// Mitsubishi GX Developer project: 12-1008_20141007   PLC: FX3U

PROGRAM MAIN
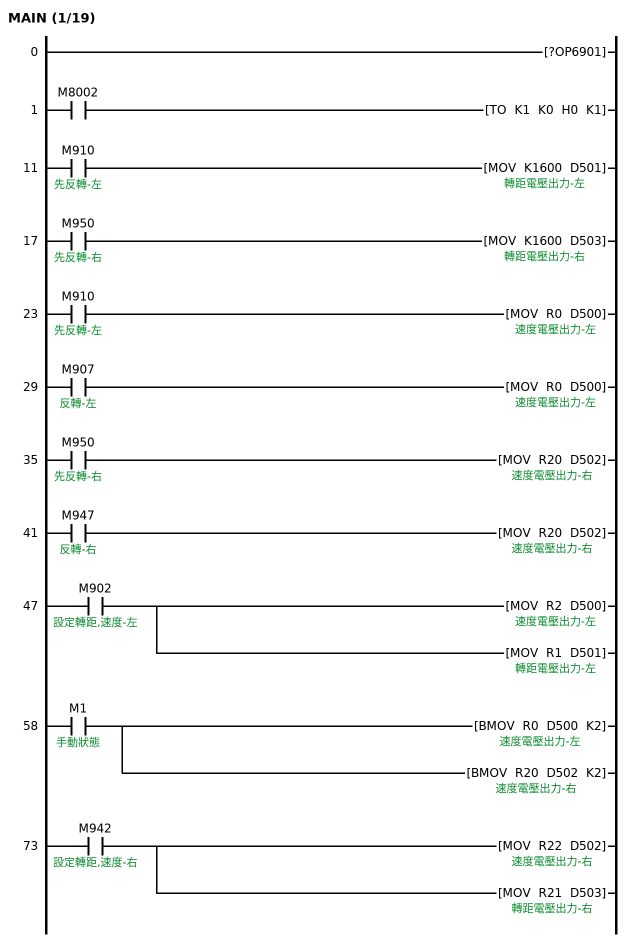
0     ?OP6901
1     LD      M8002
      TO      K1 K0 H0 K1
11    LD      M910  ; 先反轉-左
      MOV     K1600 D501  ; 轉距電壓出力-左
17    LD      M950  ; 先反轉-右
      MOV     K1600 D503  ; 轉距電壓出力-右
23    LD      M910  ; 先反轉-左
      MOV     R0 D500  ; 速度電壓出力-左
29    LD      M907  ; 反轉-左
      MOV     R0 D500
35    LD      M950  ; 先反轉-右
      MOV     R20 D502  ; 速度電壓出力-右
41    LD      M947  ; 反轉-右
      MOV     R20 D502
47    LD      M902  ; 設定轉距,速度-左
      MOV     R2 D500
      MOV     R1 D501
58    LD      M1  ; 手動狀態
      BMOV    R0 D500 K2
      BMOV    R20 D502 K2
73    LD      M942  ; 設定轉距,速度-右
      MOV     R22 D502
      MOV     R21 D503
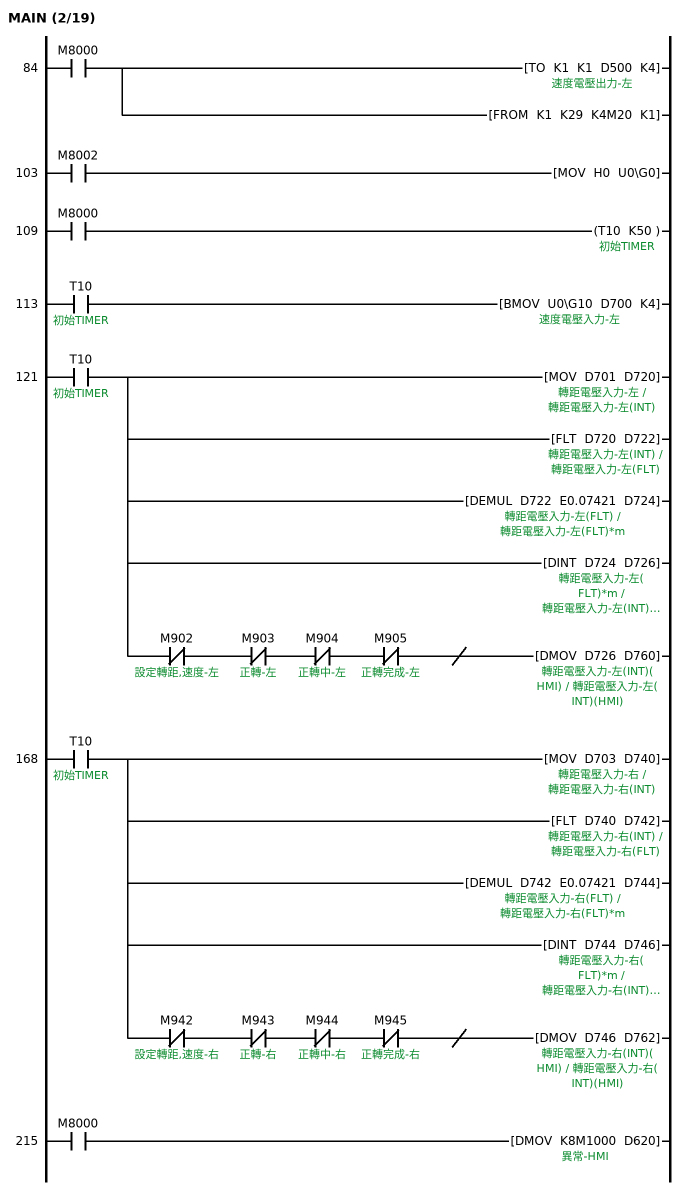
84    LD      M8000
      TO      K1 K1 D500 K4
      FROM    K1 K29 K4M20 K1  ; DA模組狀態
103   LD      M8002
      MOV     H0 U0\G0
109   LD      M8000
      OUT     T10 K50  ; 初始TIMER
113   LD      T10  ; 初始TIMER
      BMOV    U0\G10 D700 K4  ; 速度電壓入力-左
121   LD      T10  ; 初始TIMER
      MOV     D701 D720  ; 轉距電壓入力-左 / 轉距電壓入力-左(INT)
      FLT     D720 D722  ; 轉距電壓入力-左(FLT)
      DEMUL   D722 E0.07421 D724  ; 轉距電壓入力-左(FLT)*m
      DINT    D724 D726  ; 轉距電壓入力-左(INT)(HMI)
      ANI     M902  ; 設定轉距,速度-左
      ANI     M903  ; 正轉-左
      ANI     M904  ; 正轉中-左
      ANI     M905  ; 正轉完成-左
      INV
      DMOV    D726 D760  ; 轉距電壓入力-左(INT)(HMI)
168   LD      T10  ; 初始TIMER
      MOV     D703 D740  ; 轉距電壓入力-右 / 轉距電壓入力-右(INT)
      FLT     D740 D742  ; 轉距電壓入力-右(FLT)
      DEMUL   D742 E0.07421 D744  ; 轉距電壓入力-右(FLT)*m
      DINT    D744 D746  ; 轉距電壓入力-右(INT)(HMI)
      ANI     M942  ; 設定轉距,速度-右
      ANI     M943  ; 正轉-右
      ANI     M944  ; 正轉中-右
      ANI     M945  ; 正轉完成-右
      INV
      DMOV    D746 D762  ; 轉距電壓入力-右(INT)(HMI)
215   LD      M8000
      DMOV    K8M1000 D620  ; 滿料異常 / 異常-HMI
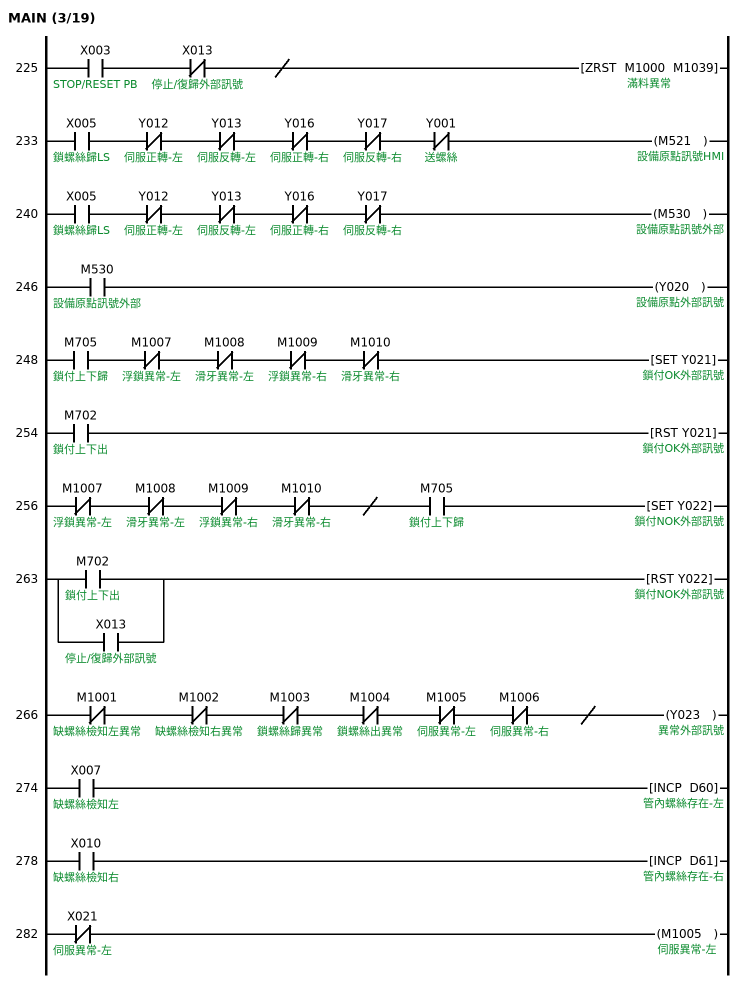
225   LD      X003  ; STOP/RESET PB
      ANI     X013  ; 停止/復歸外部訊號
      INV
      ZRST    M1000 M1039
233   LD      X005  ; 鎖螺絲歸LS
      ANI     Y012  ; 伺服正轉-左
      ANI     Y013  ; 伺服反轉-左
      ANI     Y016  ; 伺服正轉-右
      ANI     Y017  ; 伺服反轉-右
      ANI     Y001  ; 送螺絲
      OUT     M521  ; 設備原點訊號HMI
240   LD      X005  ; 鎖螺絲歸LS
      ANI     Y012  ; 伺服正轉-左
      ANI     Y013  ; 伺服反轉-左
      ANI     Y016  ; 伺服正轉-右
      ANI     Y017  ; 伺服反轉-右
      OUT     M530  ; 設備原點訊號外部
246   LD      M530  ; 設備原點訊號外部
      OUT     Y020  ; 設備原點外部訊號
248   LD      M705  ; 鎖付上下歸
      ANI     M1007  ; 浮鎖異常-左
      ANI     M1008  ; 滑牙異常-左
      ANI     M1009  ; 浮鎖異常-右
      ANI     M1010  ; 滑牙異常-右
      SET     Y021  ; 鎖付OK外部訊號
254   LD      M702  ; 鎖付上下出
      RST     Y021  ; 鎖付OK外部訊號
256   LDI     M1007  ; 浮鎖異常-左
      ANI     M1008  ; 滑牙異常-左
      ANI     M1009  ; 浮鎖異常-右
      ANI     M1010  ; 滑牙異常-右
      INV
      AND     M705  ; 鎖付上下歸
      SET     Y022  ; 鎖付NOK外部訊號
263   LD      M702  ; 鎖付上下出
      OR      X013  ; 停止/復歸外部訊號
      RST     Y022  ; 鎖付NOK外部訊號
266   LDI     M1001  ; 缺螺絲檢知左異常
      ANI     M1002  ; 缺螺絲檢知右異常
      ANI     M1003  ; 鎖螺絲歸異常
      ANI     M1004  ; 鎖螺絲出異常
      ANI     M1005  ; 伺服異常-左
      ANI     M1006  ; 伺服異常-右
      INV
      OUT     Y023  ; 異常外部訊號
274   LD      X007  ; 缺螺絲檢知左
      INCP    D60  ; 管內螺絲存在-左
278   LD      X010  ; 缺螺絲檢知右
      INCP    D61  ; 管內螺絲存在-右
282   LDI     X021  ; 伺服異常-左
      OUT     M1005  ; 伺服異常-左
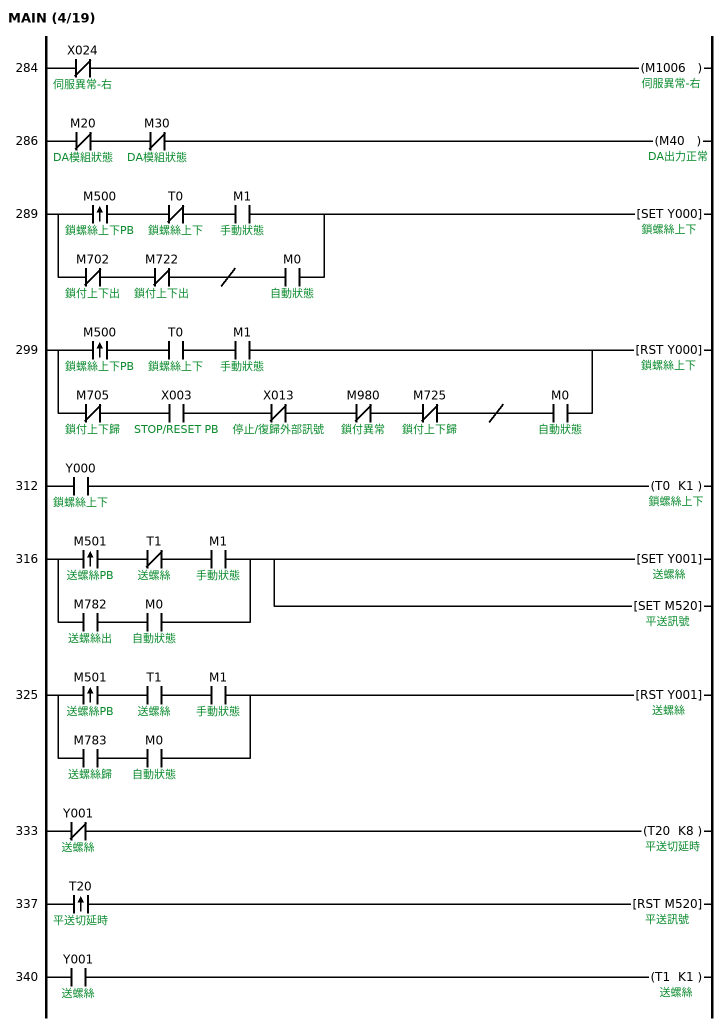
284   LDI     X024  ; 伺服異常-右
      OUT     M1006  ; 伺服異常-右
286   LDI     M20  ; DA模組狀態
      ANI     M30  ; DA模組狀態
      OUT     M40  ; DA出力正常
289   LDP     M500  ; 鎖螺絲上下PB
      ANI     T0  ; 鎖螺絲上下
      AND     M1  ; 手動狀態
      LDI     M702  ; 鎖付上下出
      ANI     M722  ; 鎖付上下出
      INV
      AND     M0  ; 自動狀態
      ORB
      SET     Y000  ; 鎖螺絲上下
299   LDP     M500  ; 鎖螺絲上下PB
      AND     T0  ; 鎖螺絲上下
      AND     M1  ; 手動狀態
      LDI     M705  ; 鎖付上下歸
      AND     X003  ; STOP/RESET PB
      ANI     X013  ; 停止/復歸外部訊號
      ANI     M980  ; 鎖付異常
      ANI     M725  ; 鎖付上下歸
      INV
      AND     M0  ; 自動狀態
      ORB
      RST     Y000  ; 鎖螺絲上下
312   LD      Y000  ; 鎖螺絲上下
      OUT     T0 K1  ; 鎖螺絲上下
316   LDP     M501  ; 送螺絲PB
      ANI     T1  ; 送螺絲
      AND     M1  ; 手動狀態
      LD      M782  ; 送螺絲出
      AND     M0  ; 自動狀態
      ORB
      SET     Y001  ; 送螺絲
      SET     M520  ; 平送訊號
325   LDP     M501  ; 送螺絲PB
      AND     T1  ; 送螺絲
      AND     M1  ; 手動狀態
      LD      M783  ; 送螺絲歸
      AND     M0  ; 自動狀態
      ORB
      RST     Y001  ; 送螺絲
333   LDI     Y001  ; 送螺絲
      OUT     T20 K8  ; 平送切延時
337   LDP     T20  ; 平送切延時
      RST     M520  ; 平送訊號
340   LD      Y001  ; 送螺絲
      OUT     T1 K1  ; 送螺絲
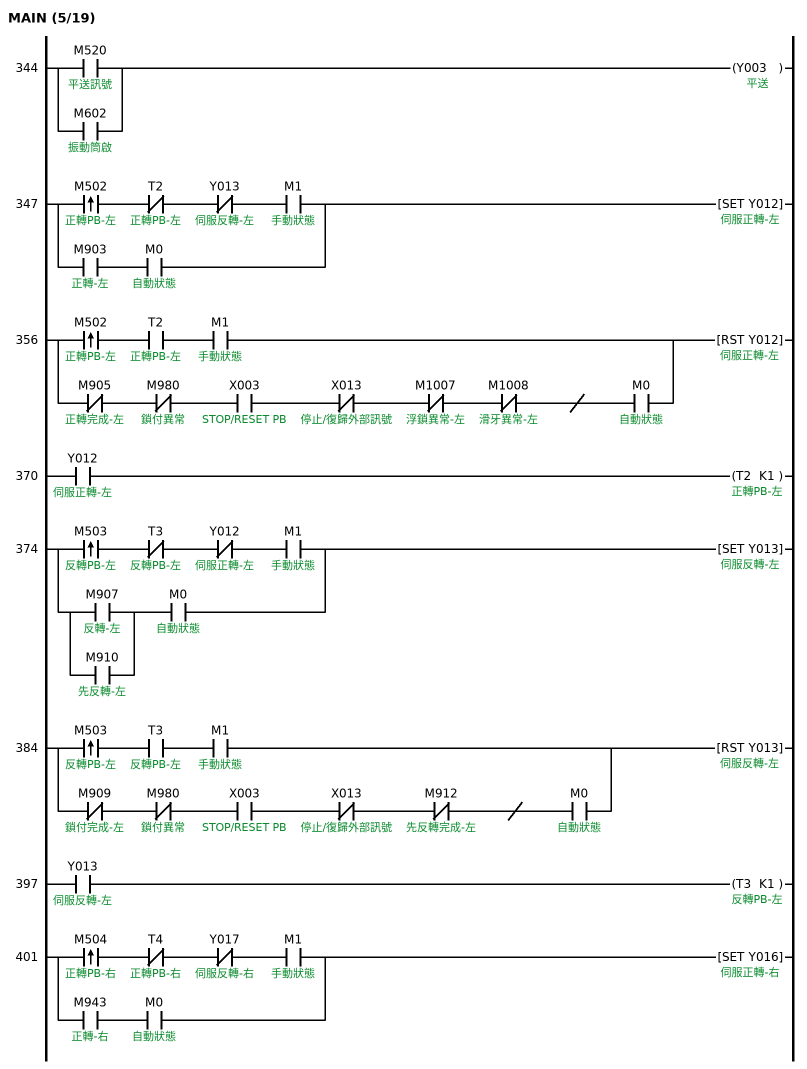
344   LD      M520  ; 平送訊號
      OR      M602  ; 振動筒啟
      OUT     Y003  ; 平送
347   LDP     M502  ; 正轉PB-左
      ANI     T2  ; 正轉PB-左
      ANI     Y013  ; 伺服反轉-左
      AND     M1  ; 手動狀態
      LD      M903  ; 正轉-左
      AND     M0  ; 自動狀態
      ORB
      SET     Y012  ; 伺服正轉-左
356   LDP     M502  ; 正轉PB-左
      AND     T2  ; 正轉PB-左
      AND     M1  ; 手動狀態
      LDI     M905  ; 正轉完成-左
      ANI     M980  ; 鎖付異常
      AND     X003  ; STOP/RESET PB
      ANI     X013  ; 停止/復歸外部訊號
      ANI     M1007  ; 浮鎖異常-左
      ANI     M1008  ; 滑牙異常-左
      INV
      AND     M0  ; 自動狀態
      ORB
      RST     Y012  ; 伺服正轉-左
370   LD      Y012  ; 伺服正轉-左
      OUT     T2 K1  ; 正轉PB-左
374   LDP     M503  ; 反轉PB-左
      ANI     T3  ; 反轉PB-左
      ANI     Y012  ; 伺服正轉-左
      AND     M1  ; 手動狀態
      LD      M907  ; 反轉-左
      OR      M910  ; 先反轉-左
      AND     M0  ; 自動狀態
      ORB
      SET     Y013  ; 伺服反轉-左
384   LDP     M503  ; 反轉PB-左
      AND     T3  ; 反轉PB-左
      AND     M1  ; 手動狀態
      LDI     M909  ; 鎖付完成-左
      ANI     M980  ; 鎖付異常
      AND     X003  ; STOP/RESET PB
      ANI     X013  ; 停止/復歸外部訊號
      ANI     M912  ; 先反轉完成-左
      INV
      AND     M0  ; 自動狀態
      ORB
      RST     Y013  ; 伺服反轉-左
397   LD      Y013  ; 伺服反轉-左
      OUT     T3 K1  ; 反轉PB-左
401   LDP     M504  ; 正轉PB-右
      ANI     T4  ; 正轉PB-右
      ANI     Y017  ; 伺服反轉-右
      AND     M1  ; 手動狀態
      LD      M943  ; 正轉-右
      AND     M0  ; 自動狀態
      ORB
      SET     Y016  ; 伺服正轉-右
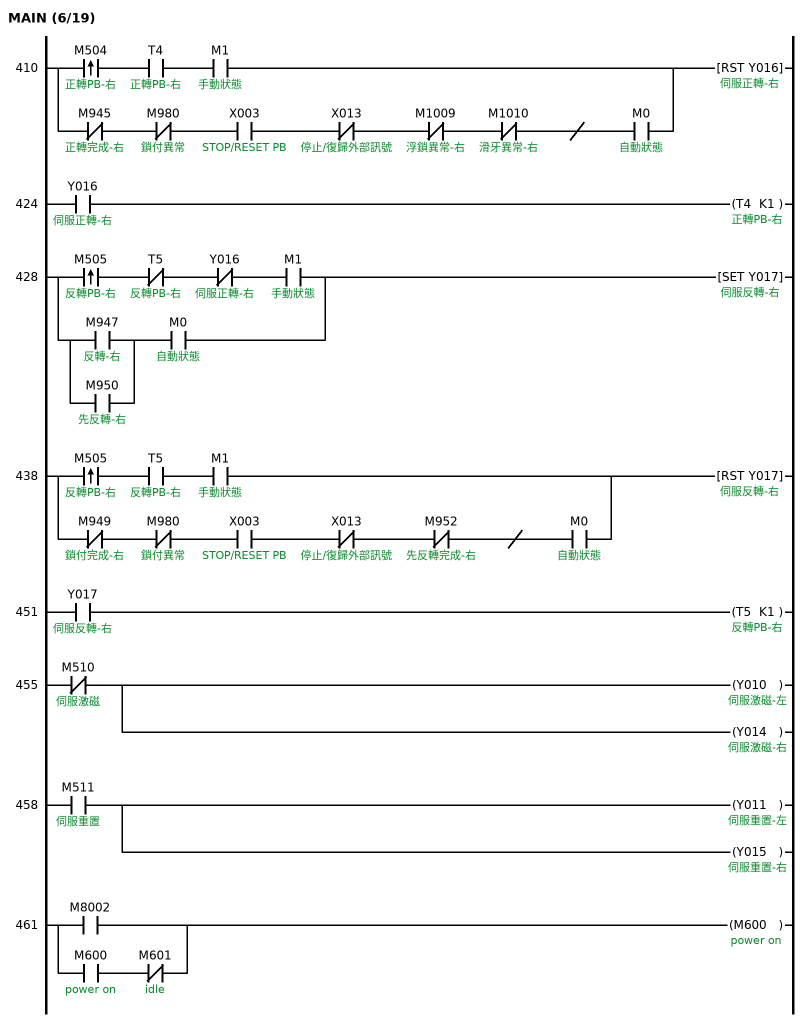
410   LDP     M504  ; 正轉PB-右
      AND     T4  ; 正轉PB-右
      AND     M1  ; 手動狀態
      LDI     M945  ; 正轉完成-右
      ANI     M980  ; 鎖付異常
      AND     X003  ; STOP/RESET PB
      ANI     X013  ; 停止/復歸外部訊號
      ANI     M1009  ; 浮鎖異常-右
      ANI     M1010  ; 滑牙異常-右
      INV
      AND     M0  ; 自動狀態
      ORB
      RST     Y016  ; 伺服正轉-右
424   LD      Y016  ; 伺服正轉-右
      OUT     T4 K1  ; 正轉PB-右
428   LDP     M505  ; 反轉PB-右
      ANI     T5  ; 反轉PB-右
      ANI     Y016  ; 伺服正轉-右
      AND     M1  ; 手動狀態
      LD      M947  ; 反轉-右
      OR      M950  ; 先反轉-右
      AND     M0  ; 自動狀態
      ORB
      SET     Y017  ; 伺服反轉-右
438   LDP     M505  ; 反轉PB-右
      AND     T5  ; 反轉PB-右
      AND     M1  ; 手動狀態
      LDI     M949  ; 鎖付完成-右
      ANI     M980  ; 鎖付異常
      AND     X003  ; STOP/RESET PB
      ANI     X013  ; 停止/復歸外部訊號
      ANI     M952  ; 先反轉完成-右
      INV
      AND     M0  ; 自動狀態
      ORB
      RST     Y017  ; 伺服反轉-右
451   LD      Y017  ; 伺服反轉-右
      OUT     T5 K1  ; 反轉PB-右
455   LDI     M510  ; 伺服激磁
      OUT     Y010  ; 伺服激磁-左
      OUT     Y014  ; 伺服激磁-右
458   LD      M511  ; 伺服重置
      OUT     Y011  ; 伺服重置-左
      OUT     Y015  ; 伺服重置-右
461   LD      M8002
      LD      M600  ; power on
      ANI     M601  ; idle
      ORB
      OUT     M600  ; power on
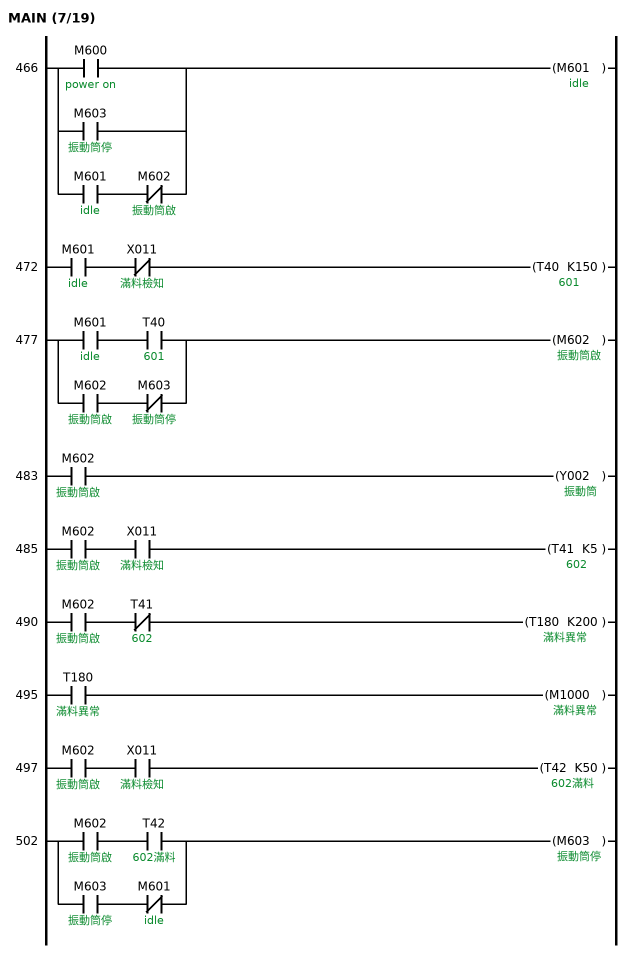
466   LD      M600  ; power on
      OR      M603  ; 振動筒停
      LD      M601  ; idle
      ANI     M602  ; 振動筒啟
      ORB
      OUT     M601  ; idle
472   LD      M601  ; idle
      ANI     X011  ; 滿料檢知
      OUT     T40 K150  ; 601
477   LD      M601  ; idle
      AND     T40  ; 601
      LD      M602  ; 振動筒啟
      ANI     M603  ; 振動筒停
      ORB
      OUT     M602  ; 振動筒啟
483   LD      M602  ; 振動筒啟
      OUT     Y002  ; 振動筒
485   LD      M602  ; 振動筒啟
      AND     X011  ; 滿料檢知
      OUT     T41 K5  ; 602
490   LD      M602  ; 振動筒啟
      ANI     T41  ; 602
      OUT     T180 K200  ; 滿料異常
495   LD      T180  ; 滿料異常
      OUT     M1000  ; 滿料異常
497   LD      M602  ; 振動筒啟
      AND     X011  ; 滿料檢知
      OUT     T42 K50  ; 602滿料
502   LD      M602  ; 振動筒啟
      AND     T42  ; 602滿料
      LD      M603  ; 振動筒停
      ANI     M601  ; idle
      ORB
      OUT     M603  ; 振動筒停
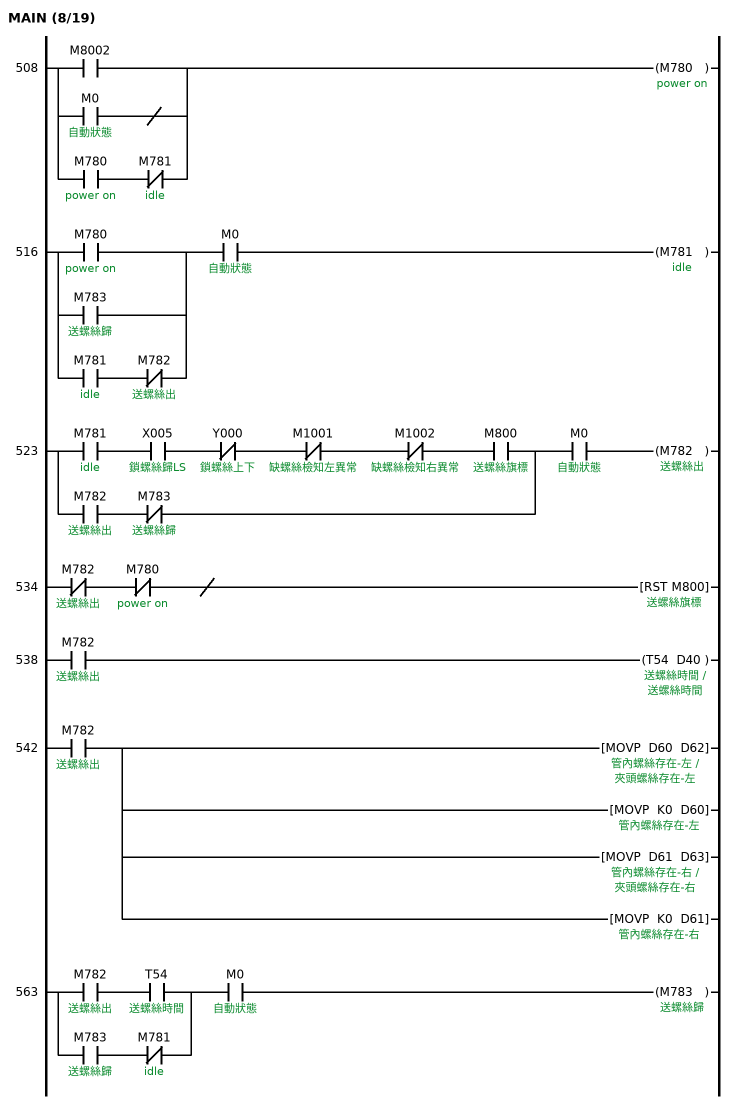
508   LD      M8002
      LD      M0  ; 自動狀態
      INV
      ORB
      LD      M780  ; power on
      ANI     M781  ; idle
      ORB
      OUT     M780  ; power on
516   LD      M780  ; power on
      OR      M783  ; 送螺絲歸
      LD      M781  ; idle
      ANI     M782  ; 送螺絲出
      ORB
      AND     M0  ; 自動狀態
      OUT     M781  ; idle
523   LD      M781  ; idle
      AND     X005  ; 鎖螺絲歸LS
      ANI     Y000  ; 鎖螺絲上下
      ANI     M1001  ; 缺螺絲檢知左異常
      ANI     M1002  ; 缺螺絲檢知右異常
      AND     M800  ; 送螺絲旗標
      LD      M782  ; 送螺絲出
      ANI     M783  ; 送螺絲歸
      ORB
      AND     M0  ; 自動狀態
      OUT     M782  ; 送螺絲出
534   LDI     M782  ; 送螺絲出
      ANI     M780  ; power on
      INV
      RST     M800  ; 送螺絲旗標
538   LD      M782  ; 送螺絲出
      OUT     T54 D40  ; 送螺絲時間 / 送螺絲時間
542   LD      M782  ; 送螺絲出
      MOVP    D60 D62  ; 夾頭螺絲存在-左
      MOVP    K0 D60
      MOVP    D61 D63  ; 夾頭螺絲存在-右
      MOVP    K0 D61
563   LD      M782  ; 送螺絲出
      AND     T54  ; 送螺絲時間
      LD      M783  ; 送螺絲歸
      ANI     M781  ; idle
      ORB
      AND     M0  ; 自動狀態
      OUT     M783  ; 送螺絲歸
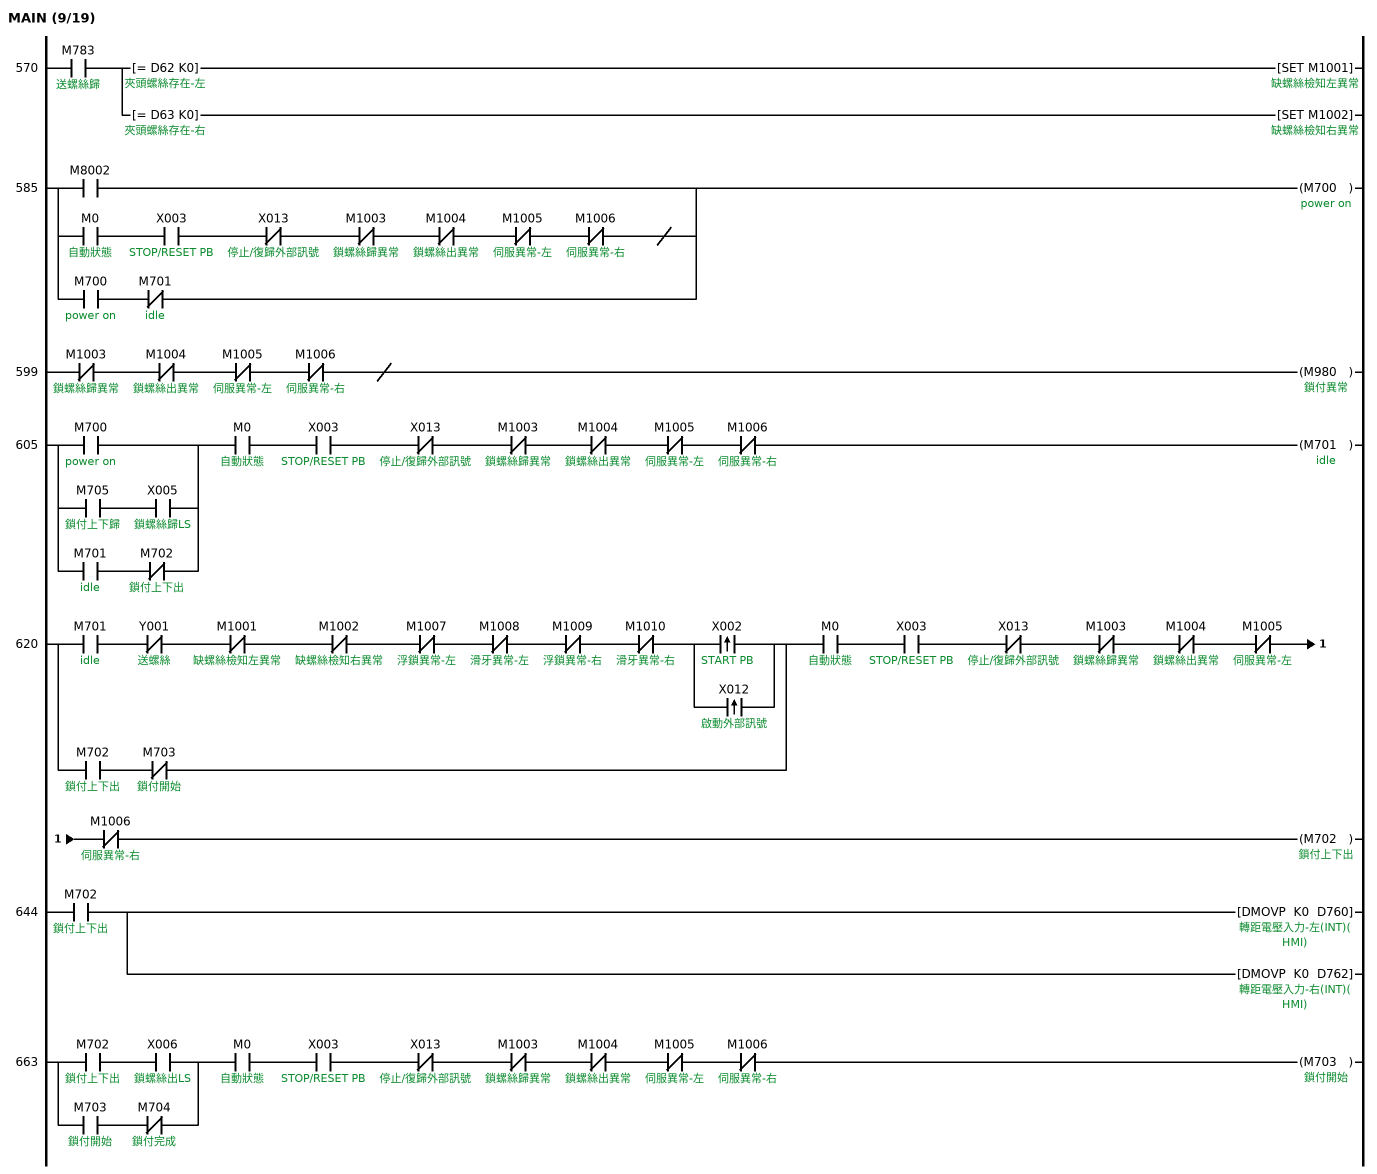
570   LD      M783  ; 送螺絲歸
      MPS
      AND=    D62 K0  ; 夾頭螺絲存在-左
      SET     M1001  ; 缺螺絲檢知左異常
      MPP
      AND=    D63 K0  ; 夾頭螺絲存在-右
      SET     M1002  ; 缺螺絲檢知右異常
585   LD      M8002
      LD      M0  ; 自動狀態
      AND     X003  ; STOP/RESET PB
      ANI     X013  ; 停止/復歸外部訊號
      ANI     M1003  ; 鎖螺絲歸異常
      ANI     M1004  ; 鎖螺絲出異常
      ANI     M1005  ; 伺服異常-左
      ANI     M1006  ; 伺服異常-右
      INV
      ORB
      LD      M700  ; power on
      ANI     M701  ; idle
      ORB
      OUT     M700  ; power on
599   LDI     M1003  ; 鎖螺絲歸異常
      ANI     M1004  ; 鎖螺絲出異常
      ANI     M1005  ; 伺服異常-左
      ANI     M1006  ; 伺服異常-右
      INV
      OUT     M980  ; 鎖付異常
605   LD      M700  ; power on
      LD      M705  ; 鎖付上下歸
      AND     X005  ; 鎖螺絲歸LS
      ORB
      LD      M701  ; idle
      ANI     M702  ; 鎖付上下出
      ORB
      AND     M0  ; 自動狀態
      AND     X003  ; STOP/RESET PB
      ANI     X013  ; 停止/復歸外部訊號
      ANI     M1003  ; 鎖螺絲歸異常
      ANI     M1004  ; 鎖螺絲出異常
      ANI     M1005  ; 伺服異常-左
      ANI     M1006  ; 伺服異常-右
      OUT     M701  ; idle
620   LD      M701  ; idle
      ANI     Y001  ; 送螺絲
      ANI     M1001  ; 缺螺絲檢知左異常
      ANI     M1002  ; 缺螺絲檢知右異常
      ANI     M1007  ; 浮鎖異常-左
      ANI     M1008  ; 滑牙異常-左
      ANI     M1009  ; 浮鎖異常-右
      ANI     M1010  ; 滑牙異常-右
      LDP     X002  ; START PB
      ORP     X012  ; 啟動外部訊號
      ANB
      LD      M702  ; 鎖付上下出
      ANI     M703  ; 鎖付開始
      ORB
      AND     M0  ; 自動狀態
      AND     X003  ; STOP/RESET PB
      ANI     X013  ; 停止/復歸外部訊號
      ANI     M1003  ; 鎖螺絲歸異常
      ANI     M1004  ; 鎖螺絲出異常
      ANI     M1005  ; 伺服異常-左
      ANI     M1006  ; 伺服異常-右
      OUT     M702  ; 鎖付上下出
644   LD      M702  ; 鎖付上下出
      DMOVP   K0 D760
      DMOVP   K0 D762
663   LD      M702  ; 鎖付上下出
      AND     X006  ; 鎖螺絲出LS
      LD      M703  ; 鎖付開始
      ANI     M704  ; 鎖付完成
      ORB
      AND     M0  ; 自動狀態
      AND     X003  ; STOP/RESET PB
      ANI     X013  ; 停止/復歸外部訊號
      ANI     M1003  ; 鎖螺絲歸異常
      ANI     M1004  ; 鎖螺絲出異常
      ANI     M1005  ; 伺服異常-左
      ANI     M1006  ; 伺服異常-右
      OUT     M703  ; 鎖付開始
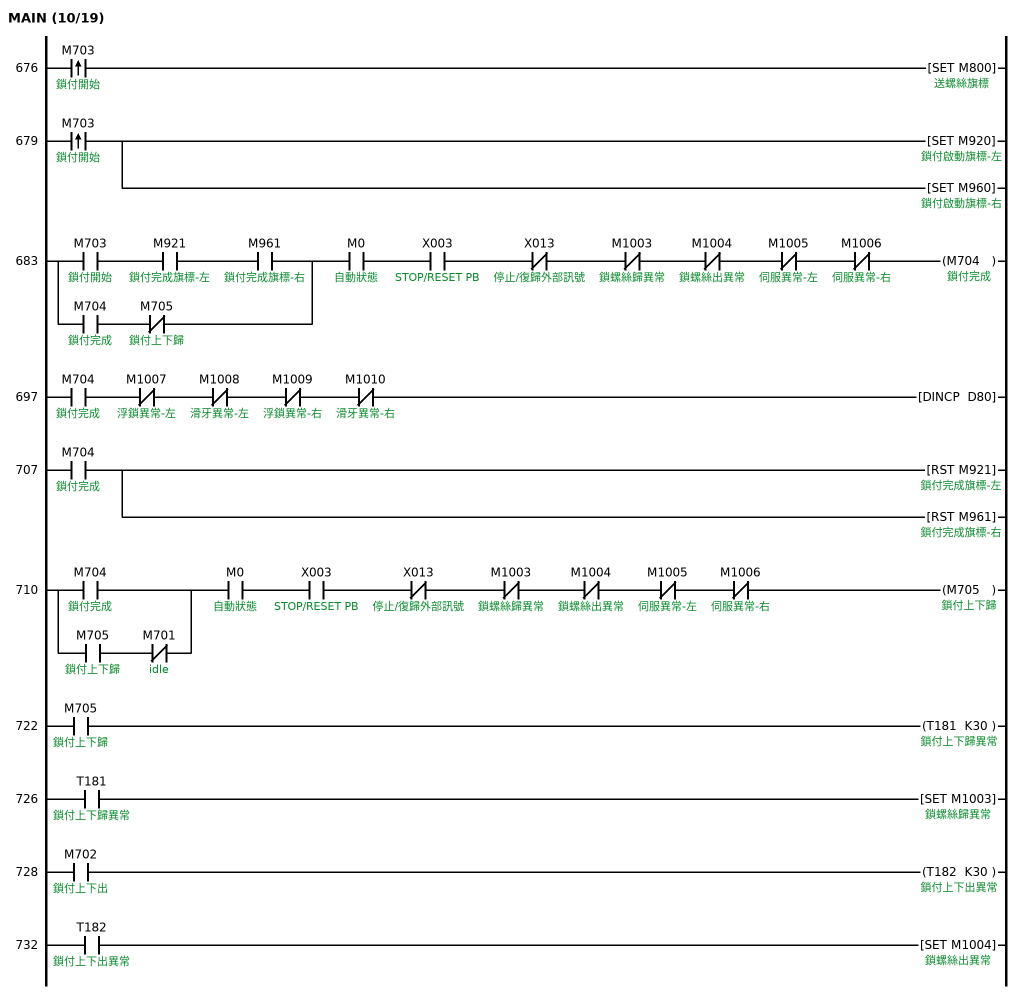
676   LDP     M703  ; 鎖付開始
      SET     M800  ; 送螺絲旗標
679   LDP     M703  ; 鎖付開始
      SET     M920  ; 鎖付啟動旗標-左
      SET     M960  ; 鎖付啟動旗標-右
683   LD      M703  ; 鎖付開始
      AND     M921  ; 鎖付完成旗標-左
      AND     M961  ; 鎖付完成旗標-右
      LD      M704  ; 鎖付完成
      ANI     M705  ; 鎖付上下歸
      ORB
      AND     M0  ; 自動狀態
      AND     X003  ; STOP/RESET PB
      ANI     X013  ; 停止/復歸外部訊號
      ANI     M1003  ; 鎖螺絲歸異常
      ANI     M1004  ; 鎖螺絲出異常
      ANI     M1005  ; 伺服異常-左
      ANI     M1006  ; 伺服異常-右
      OUT     M704  ; 鎖付完成
697   LD      M704  ; 鎖付完成
      ANI     M1007  ; 浮鎖異常-左
      ANI     M1008  ; 滑牙異常-左
      ANI     M1009  ; 浮鎖異常-右
      ANI     M1010  ; 滑牙異常-右
      DINCP   D80
707   LD      M704  ; 鎖付完成
      RST     M921  ; 鎖付完成旗標-左
      RST     M961  ; 鎖付完成旗標-右
710   LD      M704  ; 鎖付完成
      LD      M705  ; 鎖付上下歸
      ANI     M701  ; idle
      ORB
      AND     M0  ; 自動狀態
      AND     X003  ; STOP/RESET PB
      ANI     X013  ; 停止/復歸外部訊號
      ANI     M1003  ; 鎖螺絲歸異常
      ANI     M1004  ; 鎖螺絲出異常
      ANI     M1005  ; 伺服異常-左
      ANI     M1006  ; 伺服異常-右
      OUT     M705  ; 鎖付上下歸
722   LD      M705  ; 鎖付上下歸
      OUT     T181 K30  ; 鎖付上下歸異常
726   LD      T181  ; 鎖付上下歸異常
      SET     M1003  ; 鎖螺絲歸異常
728   LD      M702  ; 鎖付上下出
      OUT     T182 K30  ; 鎖付上下出異常
732   LD      T182  ; 鎖付上下出異常
      SET     M1004  ; 鎖螺絲出異常
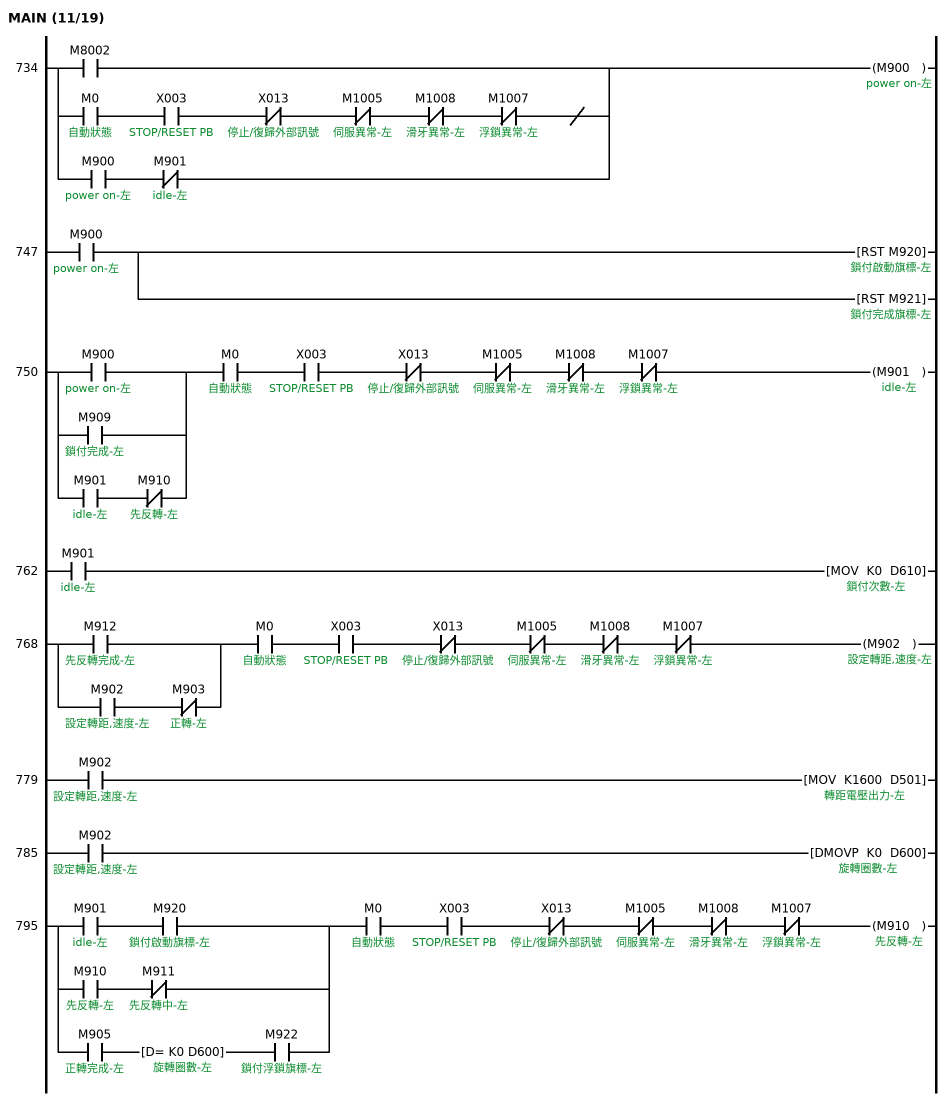
734   LD      M8002
      LD      M0  ; 自動狀態
      AND     X003  ; STOP/RESET PB
      ANI     X013  ; 停止/復歸外部訊號
      ANI     M1005  ; 伺服異常-左
      ANI     M1008  ; 滑牙異常-左
      ANI     M1007  ; 浮鎖異常-左
      INV
      ORB
      LD      M900  ; power on-左
      ANI     M901  ; idle-左
      ORB
      OUT     M900  ; power on-左
747   LD      M900  ; power on-左
      RST     M920  ; 鎖付啟動旗標-左
      RST     M921  ; 鎖付完成旗標-左
750   LD      M900  ; power on-左
      OR      M909  ; 鎖付完成-左
      LD      M901  ; idle-左
      ANI     M910  ; 先反轉-左
      ORB
      AND     M0  ; 自動狀態
      AND     X003  ; STOP/RESET PB
      ANI     X013  ; 停止/復歸外部訊號
      ANI     M1005  ; 伺服異常-左
      ANI     M1008  ; 滑牙異常-左
      ANI     M1007  ; 浮鎖異常-左
      OUT     M901  ; idle-左
762   LD      M901  ; idle-左
      MOV     K0 D610  ; 鎖付次數-左
768   LD      M912  ; 先反轉完成-左
      LD      M902  ; 設定轉距,速度-左
      ANI     M903  ; 正轉-左
      ORB
      AND     M0  ; 自動狀態
      AND     X003  ; STOP/RESET PB
      ANI     X013  ; 停止/復歸外部訊號
      ANI     M1005  ; 伺服異常-左
      ANI     M1008  ; 滑牙異常-左
      ANI     M1007  ; 浮鎖異常-左
      OUT     M902  ; 設定轉距,速度-左
779   LD      M902  ; 設定轉距,速度-左
      MOV     K1600 D501
785   LD      M902  ; 設定轉距,速度-左
      DMOVP   K0 D600  ; 旋轉圈數-左
795   LD      M901  ; idle-左
      AND     M920  ; 鎖付啟動旗標-左
      LD      M910  ; 先反轉-左
      ANI     M911  ; 先反轉中-左
      ORB
      LD      M905  ; 正轉完成-左
      ANDD=   K0 D600  ; 旋轉圈數-左
      AND     M922  ; 鎖付浮鎖旗標-左
      ORB
      AND     M0  ; 自動狀態
      AND     X003  ; STOP/RESET PB
      ANI     X013  ; 停止/復歸外部訊號
      ANI     M1005  ; 伺服異常-左
      ANI     M1008  ; 滑牙異常-左
      ANI     M1007  ; 浮鎖異常-左
      OUT     M910  ; 先反轉-左
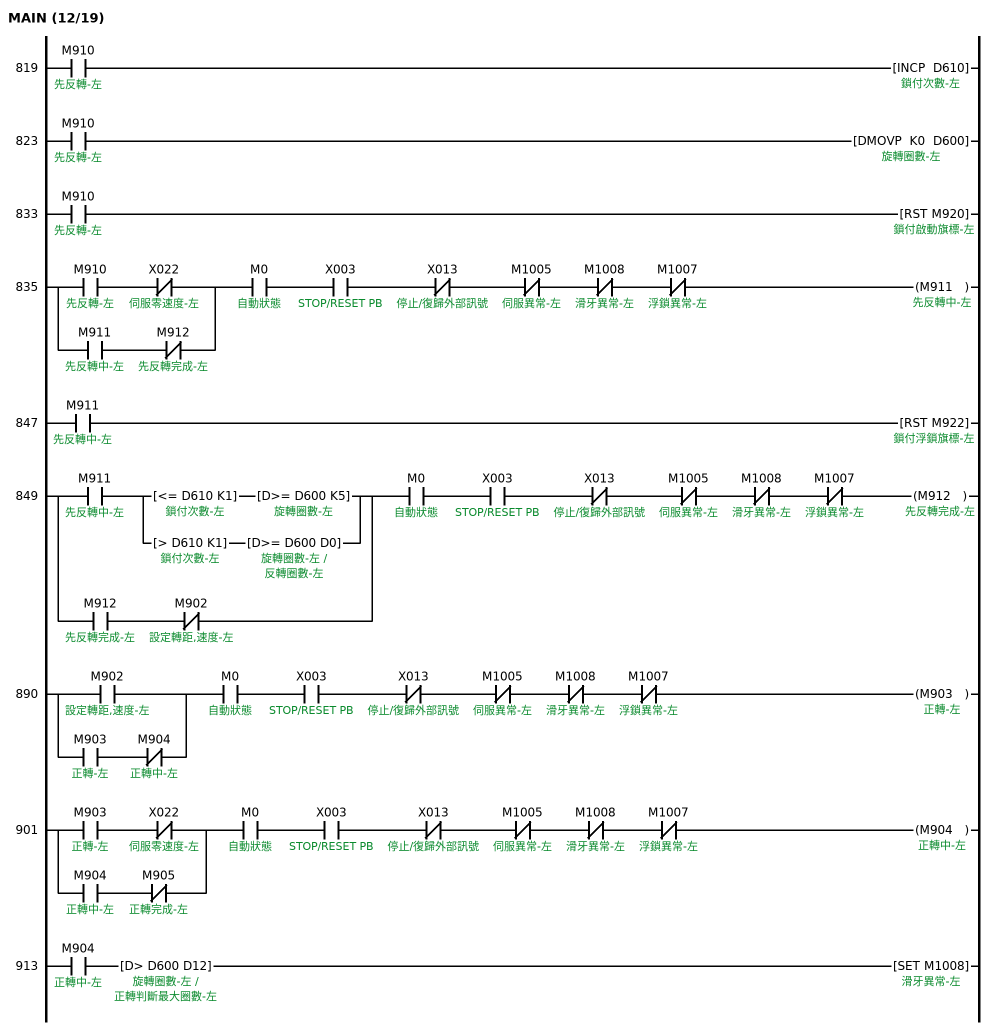
819   LD      M910  ; 先反轉-左
      INCP    D610
823   LD      M910  ; 先反轉-左
      DMOVP   K0 D600
833   LD      M910  ; 先反轉-左
      RST     M920  ; 鎖付啟動旗標-左
835   LD      M910  ; 先反轉-左
      ANI     X022  ; 伺服零速度-左
      LD      M911  ; 先反轉中-左
      ANI     M912  ; 先反轉完成-左
      ORB
      AND     M0  ; 自動狀態
      AND     X003  ; STOP/RESET PB
      ANI     X013  ; 停止/復歸外部訊號
      ANI     M1005  ; 伺服異常-左
      ANI     M1008  ; 滑牙異常-左
      ANI     M1007  ; 浮鎖異常-左
      OUT     M911  ; 先反轉中-左
847   LD      M911  ; 先反轉中-左
      RST     M922  ; 鎖付浮鎖旗標-左
849   LD      M911  ; 先反轉中-左
      LD<=    D610 K1  ; 鎖付次數-左
      ANDD>=  D600 K5  ; 旋轉圈數-左
      LD>     D610 K1  ; 鎖付次數-左
      ANDD>=  D600 D0  ; 旋轉圈數-左 / 反轉圈數-左
      ORB
      ANB
      LD      M912  ; 先反轉完成-左
      ANI     M902  ; 設定轉距,速度-左
      ORB
      AND     M0  ; 自動狀態
      AND     X003  ; STOP/RESET PB
      ANI     X013  ; 停止/復歸外部訊號
      ANI     M1005  ; 伺服異常-左
      ANI     M1008  ; 滑牙異常-左
      ANI     M1007  ; 浮鎖異常-左
      OUT     M912  ; 先反轉完成-左
890   LD      M902  ; 設定轉距,速度-左
      LD      M903  ; 正轉-左
      ANI     M904  ; 正轉中-左
      ORB
      AND     M0  ; 自動狀態
      AND     X003  ; STOP/RESET PB
      ANI     X013  ; 停止/復歸外部訊號
      ANI     M1005  ; 伺服異常-左
      ANI     M1008  ; 滑牙異常-左
      ANI     M1007  ; 浮鎖異常-左
      OUT     M903  ; 正轉-左
901   LD      M903  ; 正轉-左
      ANI     X022  ; 伺服零速度-左
      LD      M904  ; 正轉中-左
      ANI     M905  ; 正轉完成-左
      ORB
      AND     M0  ; 自動狀態
      AND     X003  ; STOP/RESET PB
      ANI     X013  ; 停止/復歸外部訊號
      ANI     M1005  ; 伺服異常-左
      ANI     M1008  ; 滑牙異常-左
      ANI     M1007  ; 浮鎖異常-左
      OUT     M904  ; 正轉中-左
913   LD      M904  ; 正轉中-左
      ANDD>   D600 D12  ; 旋轉圈數-左 / 正轉判斷最大圈數-左
      SET     M1008  ; 滑牙異常-左
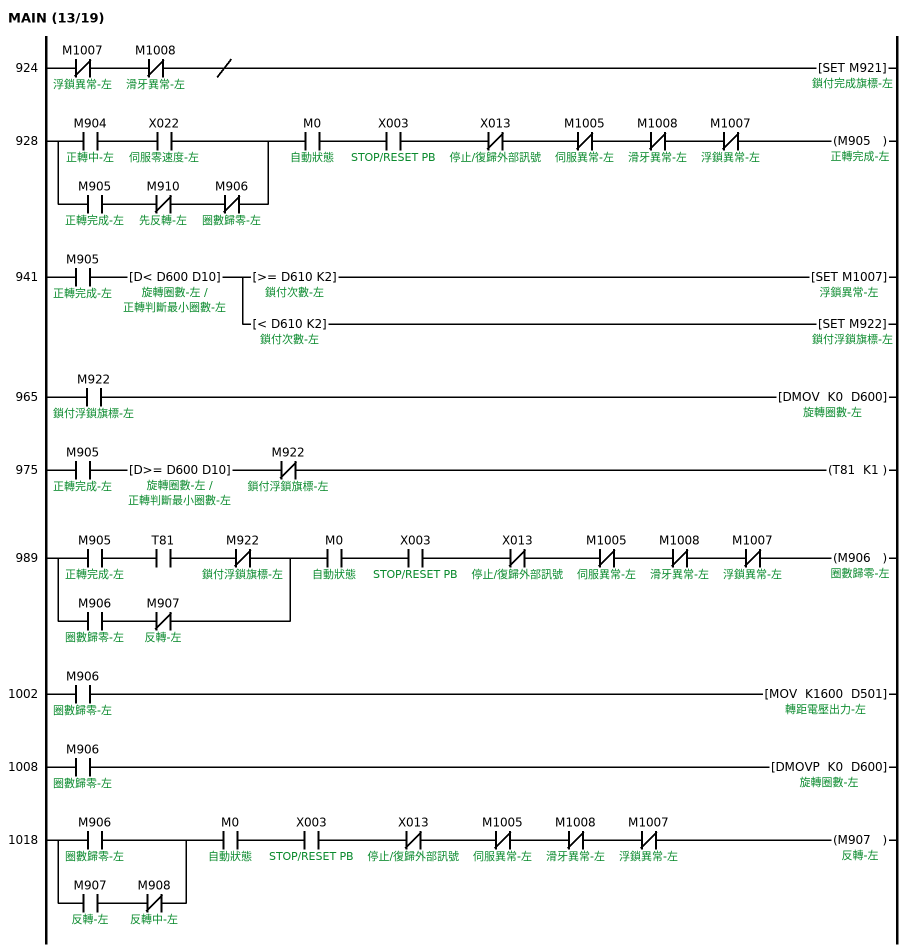
924   LDI     M1007  ; 浮鎖異常-左
      ANI     M1008  ; 滑牙異常-左
      INV
      SET     M921  ; 鎖付完成旗標-左
928   LD      M904  ; 正轉中-左
      AND     X022  ; 伺服零速度-左
      LD      M905  ; 正轉完成-左
      ANI     M910  ; 先反轉-左
      ANI     M906  ; 圈數歸零-左
      ORB
      AND     M0  ; 自動狀態
      AND     X003  ; STOP/RESET PB
      ANI     X013  ; 停止/復歸外部訊號
      ANI     M1005  ; 伺服異常-左
      ANI     M1008  ; 滑牙異常-左
      ANI     M1007  ; 浮鎖異常-左
      OUT     M905  ; 正轉完成-左
941   LD      M905  ; 正轉完成-左
      ANDD<   D600 D10  ; 旋轉圈數-左 / 正轉判斷最小圈數-左
      MPS
      AND>=   D610 K2  ; 鎖付次數-左
      SET     M1007  ; 浮鎖異常-左
      MPP
      AND<    D610 K2  ; 鎖付次數-左
      SET     M922  ; 鎖付浮鎖旗標-左
965   LD      M922  ; 鎖付浮鎖旗標-左
      DMOV    K0 D600
975   LD      M905  ; 正轉完成-左
      ANDD>=  D600 D10  ; 旋轉圈數-左 / 正轉判斷最小圈數-左
      ANI     M922  ; 鎖付浮鎖旗標-左
      OUT     T81 K1
989   LD      M905  ; 正轉完成-左
      AND     T81
      ANI     M922  ; 鎖付浮鎖旗標-左
      LD      M906  ; 圈數歸零-左
      ANI     M907  ; 反轉-左
      ORB
      AND     M0  ; 自動狀態
      AND     X003  ; STOP/RESET PB
      ANI     X013  ; 停止/復歸外部訊號
      ANI     M1005  ; 伺服異常-左
      ANI     M1008  ; 滑牙異常-左
      ANI     M1007  ; 浮鎖異常-左
      OUT     M906  ; 圈數歸零-左
1002  LD      M906  ; 圈數歸零-左
      MOV     K1600 D501
1008  LD      M906  ; 圈數歸零-左
      DMOVP   K0 D600
1018  LD      M906  ; 圈數歸零-左
      LD      M907  ; 反轉-左
      ANI     M908  ; 反轉中-左
      ORB
      AND     M0  ; 自動狀態
      AND     X003  ; STOP/RESET PB
      ANI     X013  ; 停止/復歸外部訊號
      ANI     M1005  ; 伺服異常-左
      ANI     M1008  ; 滑牙異常-左
      ANI     M1007  ; 浮鎖異常-左
      OUT     M907  ; 反轉-左
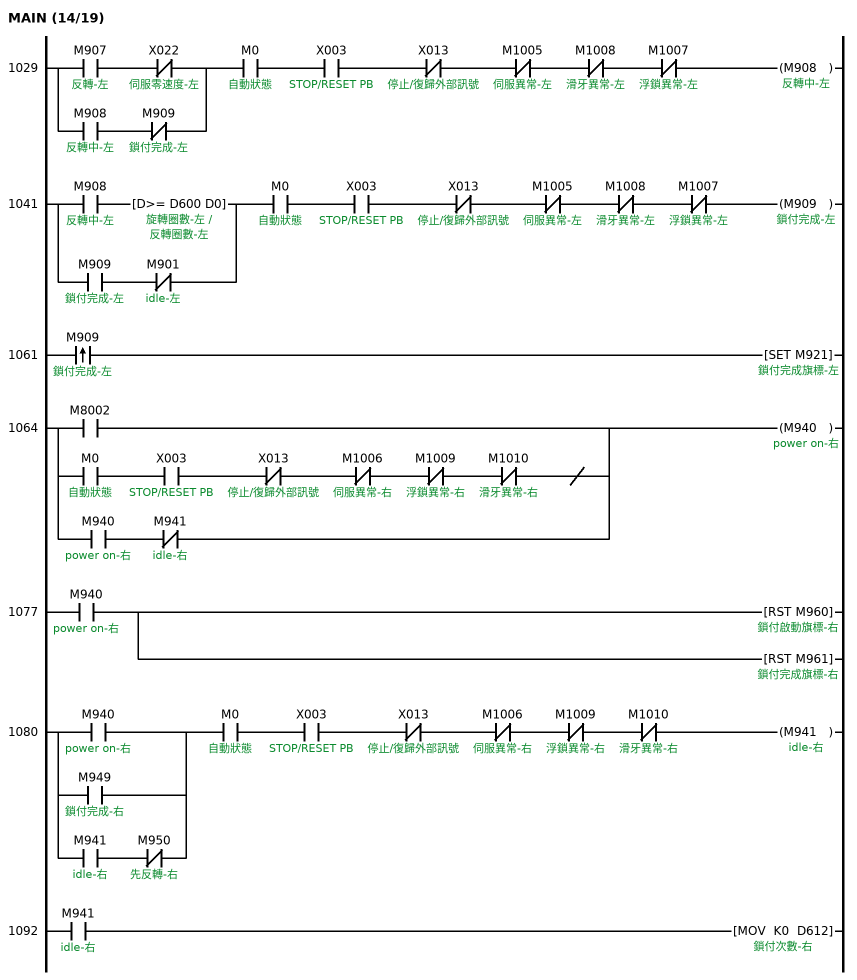
1029  LD      M907  ; 反轉-左
      ANI     X022  ; 伺服零速度-左
      LD      M908  ; 反轉中-左
      ANI     M909  ; 鎖付完成-左
      ORB
      AND     M0  ; 自動狀態
      AND     X003  ; STOP/RESET PB
      ANI     X013  ; 停止/復歸外部訊號
      ANI     M1005  ; 伺服異常-左
      ANI     M1008  ; 滑牙異常-左
      ANI     M1007  ; 浮鎖異常-左
      OUT     M908  ; 反轉中-左
1041  LD      M908  ; 反轉中-左
      ANDD>=  D600 D0  ; 旋轉圈數-左 / 反轉圈數-左
      LD      M909  ; 鎖付完成-左
      ANI     M901  ; idle-左
      ORB
      AND     M0  ; 自動狀態
      AND     X003  ; STOP/RESET PB
      ANI     X013  ; 停止/復歸外部訊號
      ANI     M1005  ; 伺服異常-左
      ANI     M1008  ; 滑牙異常-左
      ANI     M1007  ; 浮鎖異常-左
      OUT     M909  ; 鎖付完成-左
1061  LDP     M909  ; 鎖付完成-左
      SET     M921  ; 鎖付完成旗標-左
1064  LD      M8002
      LD      M0  ; 自動狀態
      AND     X003  ; STOP/RESET PB
      ANI     X013  ; 停止/復歸外部訊號
      ANI     M1006  ; 伺服異常-右
      ANI     M1009  ; 浮鎖異常-右
      ANI     M1010  ; 滑牙異常-右
      INV
      ORB
      LD      M940  ; power on-右
      ANI     M941  ; idle-右
      ORB
      OUT     M940  ; power on-右
1077  LD      M940  ; power on-右
      RST     M960  ; 鎖付啟動旗標-右
      RST     M961  ; 鎖付完成旗標-右
1080  LD      M940  ; power on-右
      OR      M949  ; 鎖付完成-右
      LD      M941  ; idle-右
      ANI     M950  ; 先反轉-右
      ORB
      AND     M0  ; 自動狀態
      AND     X003  ; STOP/RESET PB
      ANI     X013  ; 停止/復歸外部訊號
      ANI     M1006  ; 伺服異常-右
      ANI     M1009  ; 浮鎖異常-右
      ANI     M1010  ; 滑牙異常-右
      OUT     M941  ; idle-右
1092  LD      M941  ; idle-右
      MOV     K0 D612  ; 鎖付次數-右
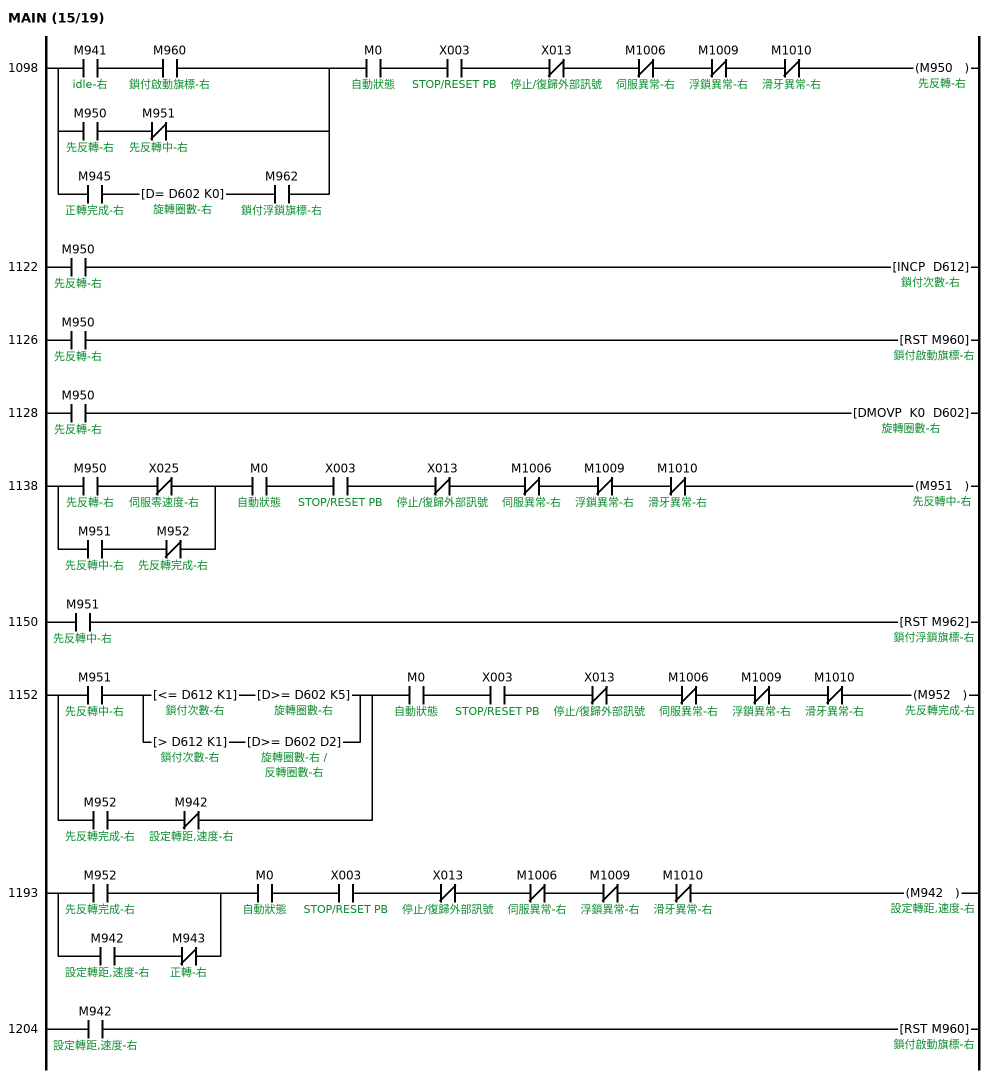
1098  LD      M941  ; idle-右
      AND     M960  ; 鎖付啟動旗標-右
      LD      M950  ; 先反轉-右
      ANI     M951  ; 先反轉中-右
      ORB
      LD      M945  ; 正轉完成-右
      ANDD=   D602 K0  ; 旋轉圈數-右
      AND     M962  ; 鎖付浮鎖旗標-右
      ORB
      AND     M0  ; 自動狀態
      AND     X003  ; STOP/RESET PB
      ANI     X013  ; 停止/復歸外部訊號
      ANI     M1006  ; 伺服異常-右
      ANI     M1009  ; 浮鎖異常-右
      ANI     M1010  ; 滑牙異常-右
      OUT     M950  ; 先反轉-右
1122  LD      M950  ; 先反轉-右
      INCP    D612
1126  LD      M950  ; 先反轉-右
      RST     M960  ; 鎖付啟動旗標-右
1128  LD      M950  ; 先反轉-右
      DMOVP   K0 D602
1138  LD      M950  ; 先反轉-右
      ANI     X025  ; 伺服零速度-右
      LD      M951  ; 先反轉中-右
      ANI     M952  ; 先反轉完成-右
      ORB
      AND     M0  ; 自動狀態
      AND     X003  ; STOP/RESET PB
      ANI     X013  ; 停止/復歸外部訊號
      ANI     M1006  ; 伺服異常-右
      ANI     M1009  ; 浮鎖異常-右
      ANI     M1010  ; 滑牙異常-右
      OUT     M951  ; 先反轉中-右
1150  LD      M951  ; 先反轉中-右
      RST     M962  ; 鎖付浮鎖旗標-右
1152  LD      M951  ; 先反轉中-右
      LD<=    D612 K1  ; 鎖付次數-右
      ANDD>=  D602 K5  ; 旋轉圈數-右
      LD>     D612 K1  ; 鎖付次數-右
      ANDD>=  D602 D2  ; 旋轉圈數-右 / 反轉圈數-右
      ORB
      ANB
      LD      M952  ; 先反轉完成-右
      ANI     M942  ; 設定轉距,速度-右
      ORB
      AND     M0  ; 自動狀態
      AND     X003  ; STOP/RESET PB
      ANI     X013  ; 停止/復歸外部訊號
      ANI     M1006  ; 伺服異常-右
      ANI     M1009  ; 浮鎖異常-右
      ANI     M1010  ; 滑牙異常-右
      OUT     M952  ; 先反轉完成-右
1193  LD      M952  ; 先反轉完成-右
      LD      M942  ; 設定轉距,速度-右
      ANI     M943  ; 正轉-右
      ORB
      AND     M0  ; 自動狀態
      AND     X003  ; STOP/RESET PB
      ANI     X013  ; 停止/復歸外部訊號
      ANI     M1006  ; 伺服異常-右
      ANI     M1009  ; 浮鎖異常-右
      ANI     M1010  ; 滑牙異常-右
      OUT     M942  ; 設定轉距,速度-右
1204  LD      M942  ; 設定轉距,速度-右
      RST     M960  ; 鎖付啟動旗標-右
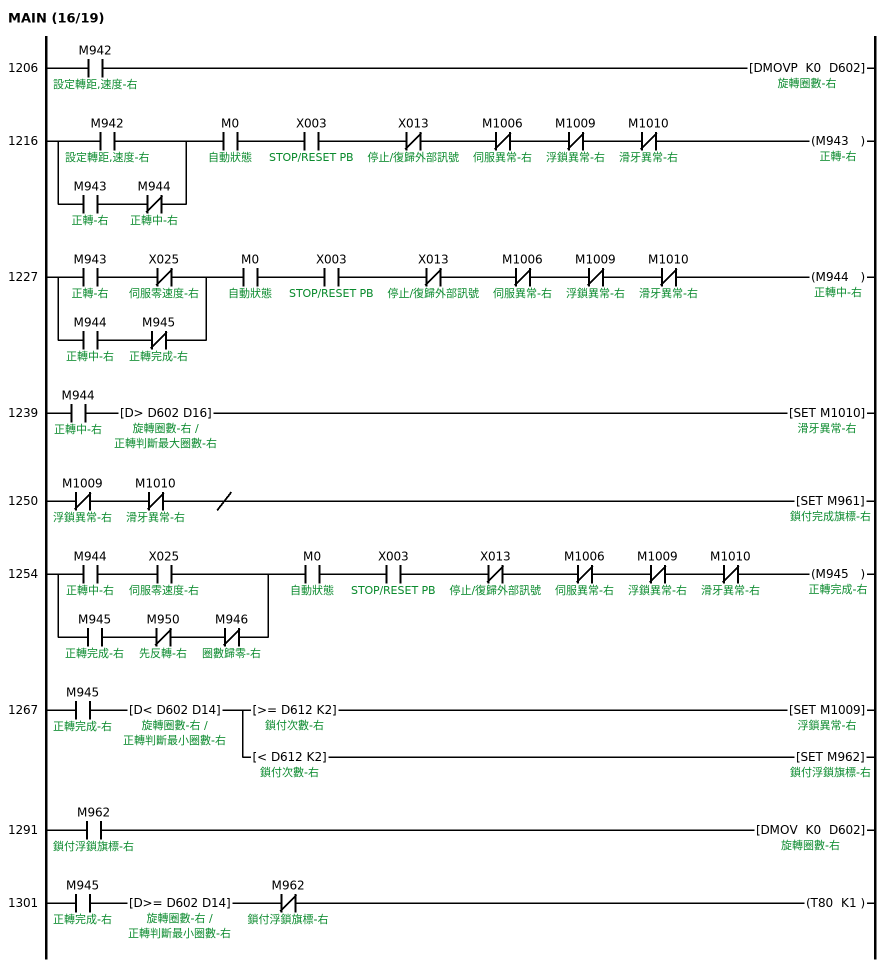
1206  LD      M942  ; 設定轉距,速度-右
      DMOVP   K0 D602
1216  LD      M942  ; 設定轉距,速度-右
      LD      M943  ; 正轉-右
      ANI     M944  ; 正轉中-右
      ORB
      AND     M0  ; 自動狀態
      AND     X003  ; STOP/RESET PB
      ANI     X013  ; 停止/復歸外部訊號
      ANI     M1006  ; 伺服異常-右
      ANI     M1009  ; 浮鎖異常-右
      ANI     M1010  ; 滑牙異常-右
      OUT     M943  ; 正轉-右
1227  LD      M943  ; 正轉-右
      ANI     X025  ; 伺服零速度-右
      LD      M944  ; 正轉中-右
      ANI     M945  ; 正轉完成-右
      ORB
      AND     M0  ; 自動狀態
      AND     X003  ; STOP/RESET PB
      ANI     X013  ; 停止/復歸外部訊號
      ANI     M1006  ; 伺服異常-右
      ANI     M1009  ; 浮鎖異常-右
      ANI     M1010  ; 滑牙異常-右
      OUT     M944  ; 正轉中-右
1239  LD      M944  ; 正轉中-右
      ANDD>   D602 D16  ; 旋轉圈數-右 / 正轉判斷最大圈數-右
      SET     M1010  ; 滑牙異常-右
1250  LDI     M1009  ; 浮鎖異常-右
      ANI     M1010  ; 滑牙異常-右
      INV
      SET     M961  ; 鎖付完成旗標-右
1254  LD      M944  ; 正轉中-右
      AND     X025  ; 伺服零速度-右
      LD      M945  ; 正轉完成-右
      ANI     M950  ; 先反轉-右
      ANI     M946  ; 圈數歸零-右
      ORB
      AND     M0  ; 自動狀態
      AND     X003  ; STOP/RESET PB
      ANI     X013  ; 停止/復歸外部訊號
      ANI     M1006  ; 伺服異常-右
      ANI     M1009  ; 浮鎖異常-右
      ANI     M1010  ; 滑牙異常-右
      OUT     M945  ; 正轉完成-右
1267  LD      M945  ; 正轉完成-右
      ANDD<   D602 D14  ; 旋轉圈數-右 / 正轉判斷最小圈數-右
      MPS
      AND>=   D612 K2  ; 鎖付次數-右
      SET     M1009  ; 浮鎖異常-右
      MPP
      AND<    D612 K2  ; 鎖付次數-右
      SET     M962  ; 鎖付浮鎖旗標-右
1291  LD      M962  ; 鎖付浮鎖旗標-右
      DMOV    K0 D602
1301  LD      M945  ; 正轉完成-右
      ANDD>=  D602 D14  ; 旋轉圈數-右 / 正轉判斷最小圈數-右
      ANI     M962  ; 鎖付浮鎖旗標-右
      OUT     T80 K1
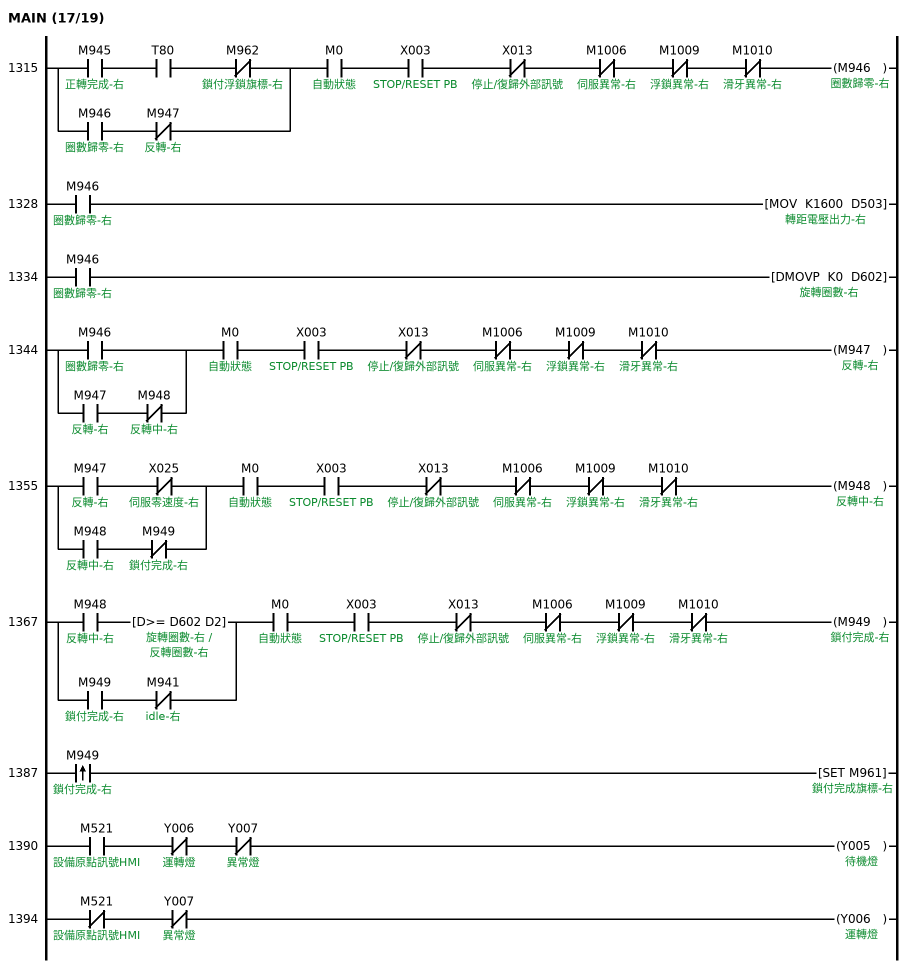
1315  LD      M945  ; 正轉完成-右
      AND     T80
      ANI     M962  ; 鎖付浮鎖旗標-右
      LD      M946  ; 圈數歸零-右
      ANI     M947  ; 反轉-右
      ORB
      AND     M0  ; 自動狀態
      AND     X003  ; STOP/RESET PB
      ANI     X013  ; 停止/復歸外部訊號
      ANI     M1006  ; 伺服異常-右
      ANI     M1009  ; 浮鎖異常-右
      ANI     M1010  ; 滑牙異常-右
      OUT     M946  ; 圈數歸零-右
1328  LD      M946  ; 圈數歸零-右
      MOV     K1600 D503
1334  LD      M946  ; 圈數歸零-右
      DMOVP   K0 D602
1344  LD      M946  ; 圈數歸零-右
      LD      M947  ; 反轉-右
      ANI     M948  ; 反轉中-右
      ORB
      AND     M0  ; 自動狀態
      AND     X003  ; STOP/RESET PB
      ANI     X013  ; 停止/復歸外部訊號
      ANI     M1006  ; 伺服異常-右
      ANI     M1009  ; 浮鎖異常-右
      ANI     M1010  ; 滑牙異常-右
      OUT     M947  ; 反轉-右
1355  LD      M947  ; 反轉-右
      ANI     X025  ; 伺服零速度-右
      LD      M948  ; 反轉中-右
      ANI     M949  ; 鎖付完成-右
      ORB
      AND     M0  ; 自動狀態
      AND     X003  ; STOP/RESET PB
      ANI     X013  ; 停止/復歸外部訊號
      ANI     M1006  ; 伺服異常-右
      ANI     M1009  ; 浮鎖異常-右
      ANI     M1010  ; 滑牙異常-右
      OUT     M948  ; 反轉中-右
1367  LD      M948  ; 反轉中-右
      ANDD>=  D602 D2  ; 旋轉圈數-右 / 反轉圈數-右
      LD      M949  ; 鎖付完成-右
      ANI     M941  ; idle-右
      ORB
      AND     M0  ; 自動狀態
      AND     X003  ; STOP/RESET PB
      ANI     X013  ; 停止/復歸外部訊號
      ANI     M1006  ; 伺服異常-右
      ANI     M1009  ; 浮鎖異常-右
      ANI     M1010  ; 滑牙異常-右
      OUT     M949  ; 鎖付完成-右
1387  LDP     M949  ; 鎖付完成-右
      SET     M961  ; 鎖付完成旗標-右
1390  LD      M521  ; 設備原點訊號HMI
      ANI     Y006  ; 運轉燈
      ANI     Y007  ; 異常燈
      OUT     Y005  ; 待機燈
1394  LDI     M521  ; 設備原點訊號HMI
      ANI     Y007  ; 異常燈
      OUT     Y006  ; 運轉燈
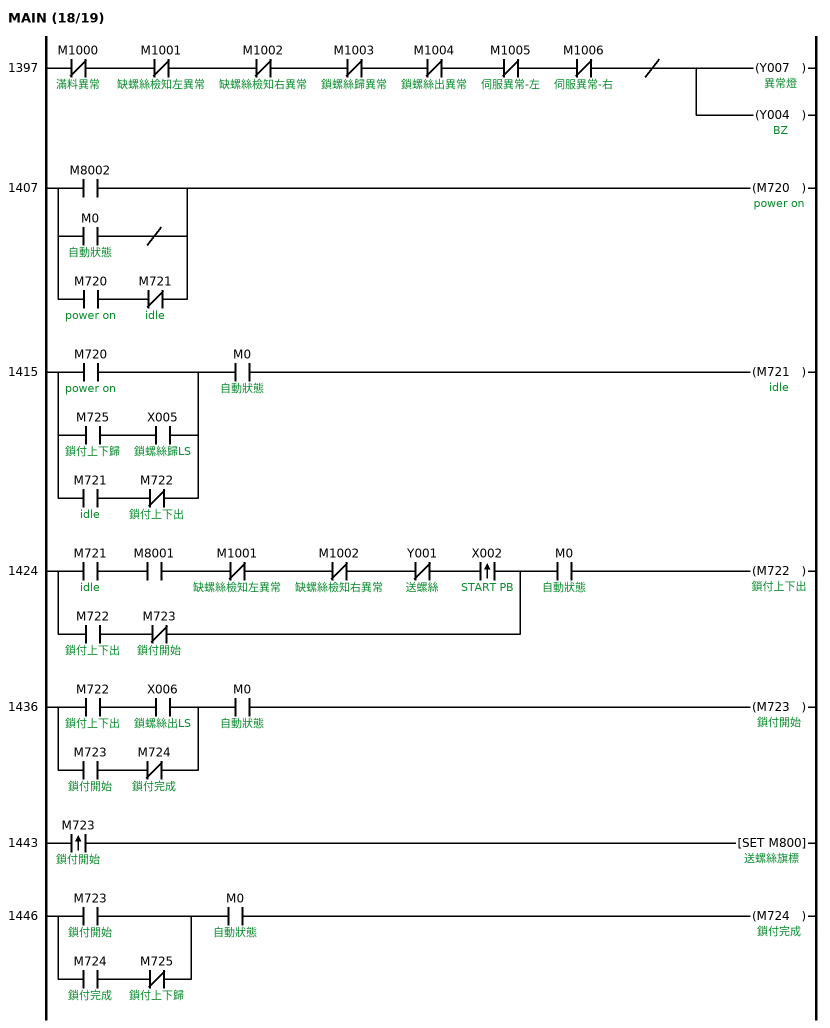
1397  LDI     M1000  ; 滿料異常
      ANI     M1001  ; 缺螺絲檢知左異常
      ANI     M1002  ; 缺螺絲檢知右異常
      ANI     M1003  ; 鎖螺絲歸異常
      ANI     M1004  ; 鎖螺絲出異常
      ANI     M1005  ; 伺服異常-左
      ANI     M1006  ; 伺服異常-右
      INV
      OUT     Y007  ; 異常燈
      OUT     Y004  ; BZ
1407  LD      M8002
      LD      M0  ; 自動狀態
      INV
      ORB
      LD      M720  ; power on
      ANI     M721  ; idle
      ORB
      OUT     M720  ; power on
1415  LD      M720  ; power on
      LD      M725  ; 鎖付上下歸
      AND     X005  ; 鎖螺絲歸LS
      ORB
      LD      M721  ; idle
      ANI     M722  ; 鎖付上下出
      ORB
      AND     M0  ; 自動狀態
      OUT     M721  ; idle
1424  LD      M721  ; idle
      AND     M8001
      ANI     M1001  ; 缺螺絲檢知左異常
      ANI     M1002  ; 缺螺絲檢知右異常
      ANI     Y001  ; 送螺絲
      ANDP    X002  ; START PB
      LD      M722  ; 鎖付上下出
      ANI     M723  ; 鎖付開始
      ORB
      AND     M0  ; 自動狀態
      OUT     M722  ; 鎖付上下出
1436  LD      M722  ; 鎖付上下出
      AND     X006  ; 鎖螺絲出LS
      LD      M723  ; 鎖付開始
      ANI     M724  ; 鎖付完成
      ORB
      AND     M0  ; 自動狀態
      OUT     M723  ; 鎖付開始
1443  LDP     M723  ; 鎖付開始
      SET     M800  ; 送螺絲旗標
1446  LD      M723  ; 鎖付開始
      LD      M724  ; 鎖付完成
      ANI     M725  ; 鎖付上下歸
      ORB
      AND     M0  ; 自動狀態
      OUT     M724  ; 鎖付完成
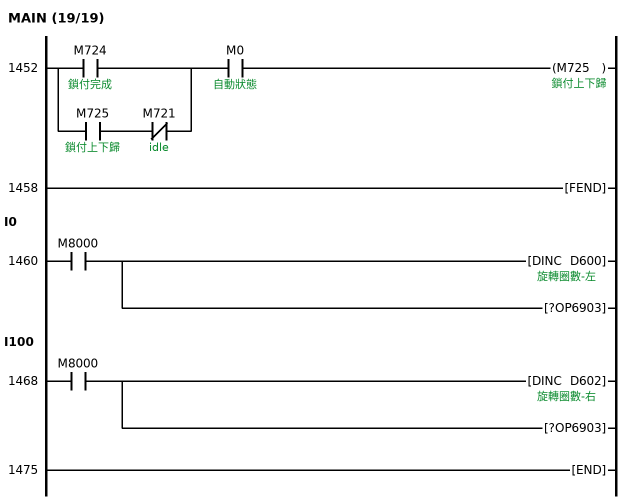
1452  LD      M724  ; 鎖付完成
      LD      M725  ; 鎖付上下歸
      ANI     M721  ; idle
      ORB
      AND     M0  ; 自動狀態
      OUT     M725  ; 鎖付上下歸
1458  FEND
      I0
1460  LD      M8000
      DINC    D600
      ?OP6903
      I100
1468  LD      M8000
      DINC    D602
      ?OP6903
1475  END
END_PROGRAM

// device comments not shown above
X000  ; Z相左
X001  ; Z相右
X020  ; 伺服準備-左
X023  ; 伺服準備-右
D200  ; 1反轉圈數-左
D202  ; 1反轉圈數-右
D601  ; **********
D603  ; **********
D621  ; 異常-HMI
D702  ; 速度電壓入力-右
D723  ; ***************
D743  ; ***************
R40  ; 手動速度
R41  ; 手動轉距
T53  ; 送螺絲TEST
